Staubli VAL3: _WaitPart.pgx

public program _WaitPart()
// Wait part made in machine and mould fully open
begin
  //!brief
  // Wait for a part being made and conditions for the robot to enter mold.
  //
  call WaitPart(false)
end
